(* Logix 5000 project; controller Joltek_RA_5069PLC002 vendor 1 type 14 code 226 rev 34.15; software revision 34.04; part 2 of 3 *)
(* tags used below, declared in another part *)
   CapperData : UDT_MachineData;
   CasePackerData : UDT_MachineData;
   FillerData : UDT_MachineData;
   LabelerData : UDT_MachineData;
   PalletizerData : UDT_MachineData;
   shiftHour : INT;
   HMI_INT : INT[100];
   HMI_REAL : REAL[100];
   Sys_DINT : DINT[100];
   Sys_FIFO_C : CONTROL[50];
   Sys_Timer : TIMER[100];
   System_Date_Time : DINT[7];
(* MainProgram, continued *)

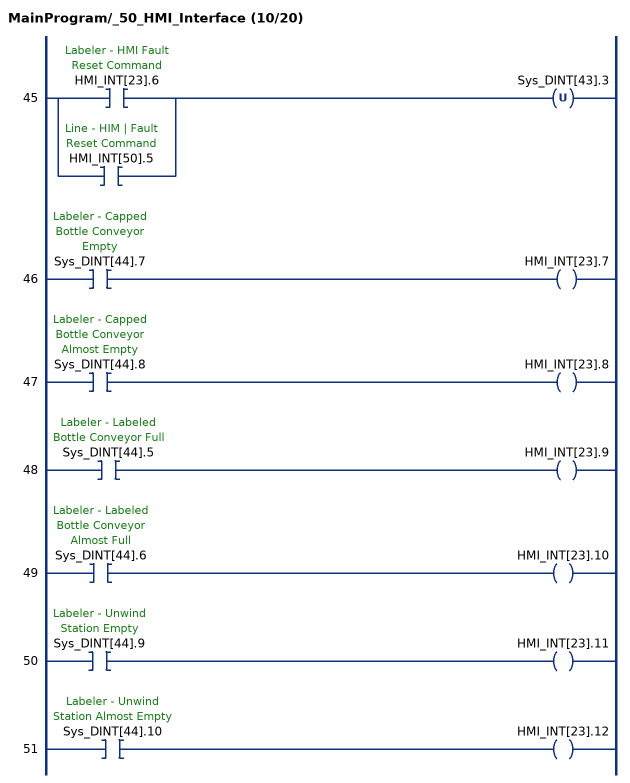
   45: [XIC(HMI_INT[23].6) ,XIC(HMI_INT[50].5) ]OTU(Sys_DINT[43].3);
   46: XIC(Sys_DINT[44].7)OTE(HMI_INT[23].7);
   47: XIC(Sys_DINT[44].8)OTE(HMI_INT[23].8);
   48: XIC(Sys_DINT[44].5)OTE(HMI_INT[23].9);
   49: XIC(Sys_DINT[44].6)OTE(HMI_INT[23].10);
   50: XIC(Sys_DINT[44].9)OTE(HMI_INT[23].11);
   51: XIC(Sys_DINT[44].10)OTE(HMI_INT[23].12);
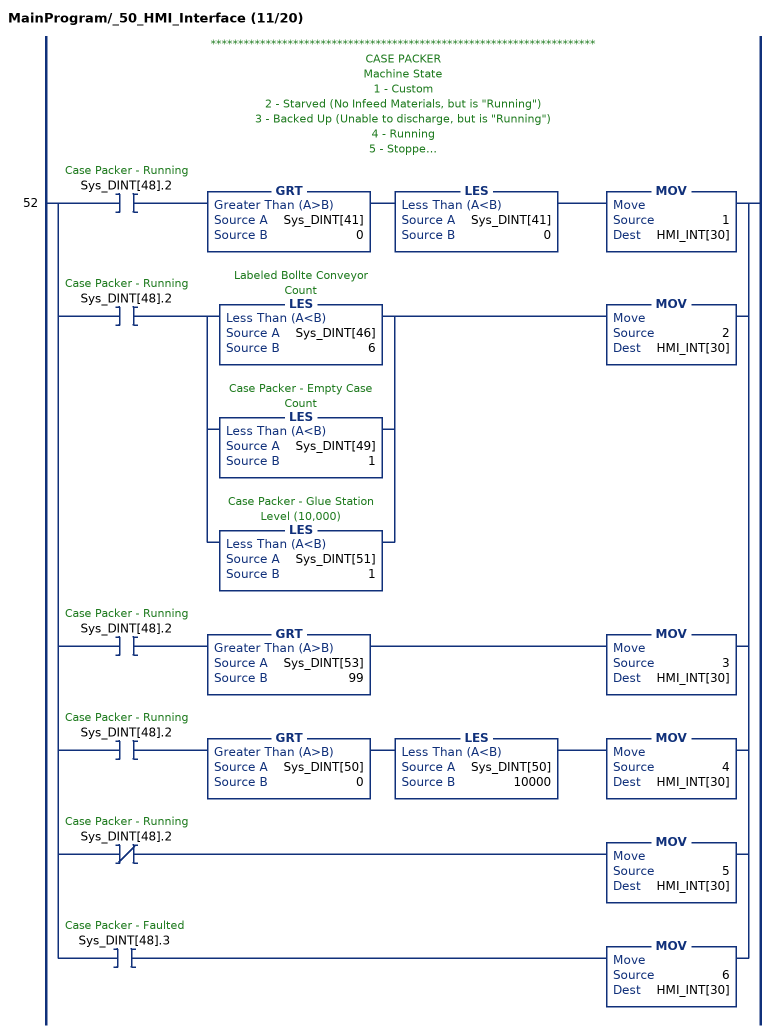
   // **********************************************************************
   // CASE PACKER
   // Machine State
   // 1 - Custom
   // 2 - Starved (No Infeed Materials, but is "Running")
   // 3 - Backed Up (Unable to discharge, but is "Running")
   // 4 - Running
   // 5 - Stopped
   // 6 - Faulted
   52: [XIC(Sys_DINT[48].2) GRT(Sys_DINT[41],0) LES(Sys_DINT[41],0) MOV(1,HMI_INT[30]) ,XIC(Sys_DINT[48].2) [LES(Sys_DINT[46],6) ,LES(Sys_DINT[49],1) ,LES(Sys_DINT[51],1) ] MOV(2,HMI_INT[30]) ,XIC(Sys_DINT[48].2) GRT(Sys_DINT[53],99) MOV(3,HMI_INT[30]) ,XIC(Sys_DINT[48].2) GRT(Sys_DINT[50],0) LES(Sys_DINT[50],10000) MOV(4,HMI_INT[30]) ,XIO(Sys_DINT[48].2) MOV(5,HMI_INT[30]) ,XIC(Sys_DINT[48].3) MOV(6,HMI_INT[30]) ];
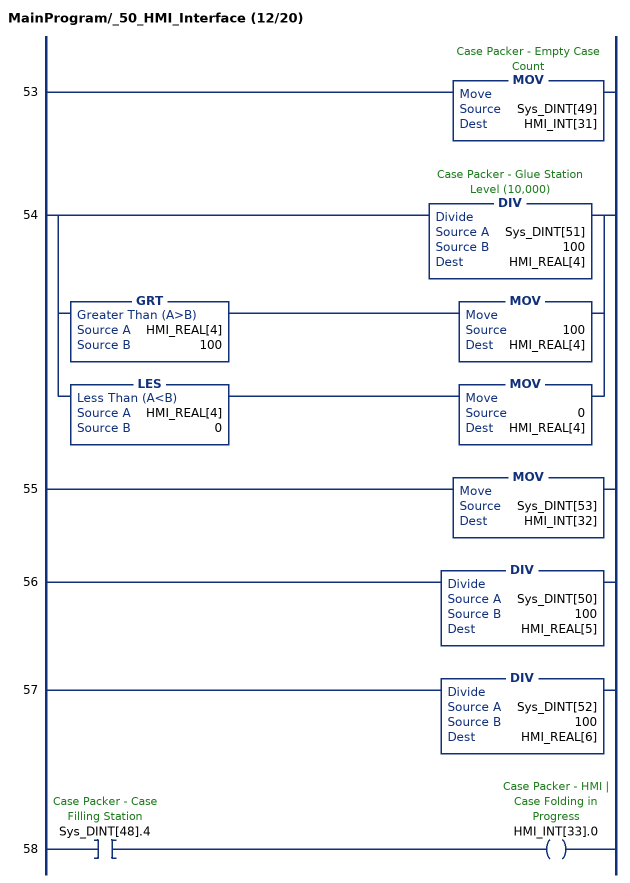
   53: MOV(Sys_DINT[49],HMI_INT[31]);
   54: [DIV(Sys_DINT[51],100,HMI_REAL[4]) ,GRT(HMI_REAL[4],100) MOV(100,HMI_REAL[4]) ,LES(HMI_REAL[4],0) MOV(0,HMI_REAL[4]) ];
   55: MOV(Sys_DINT[53],HMI_INT[32]);
   56: DIV(Sys_DINT[50],100,HMI_REAL[5]);
   57: DIV(Sys_DINT[52],100,HMI_REAL[6]);
   58: XIC(Sys_DINT[48].4)OTE(HMI_INT[33].0);
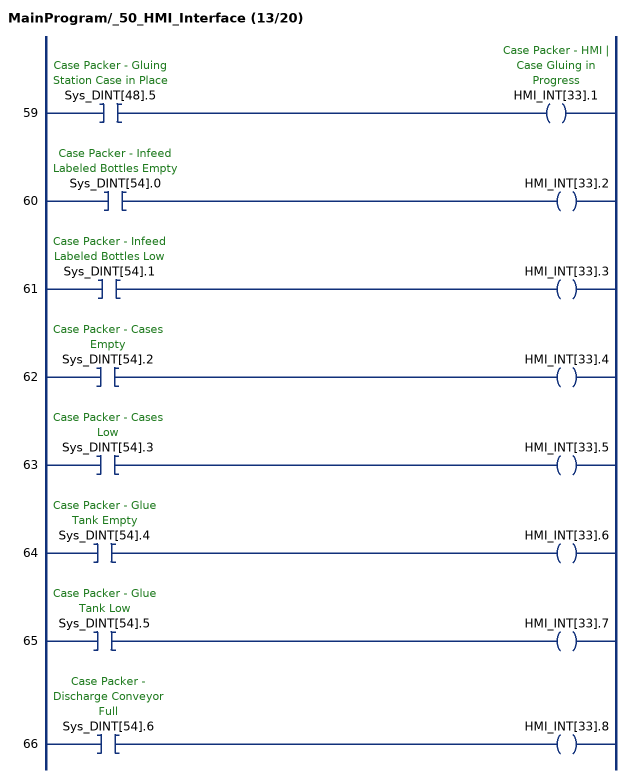
   59: XIC(Sys_DINT[48].5)OTE(HMI_INT[33].1);
   60: XIC(Sys_DINT[54].0)OTE(HMI_INT[33].2);
   61: XIC(Sys_DINT[54].1)OTE(HMI_INT[33].3);
   62: XIC(Sys_DINT[54].2)OTE(HMI_INT[33].4);
   63: XIC(Sys_DINT[54].3)OTE(HMI_INT[33].5);
   64: XIC(Sys_DINT[54].4)OTE(HMI_INT[33].6);
   65: XIC(Sys_DINT[54].5)OTE(HMI_INT[33].7);
   66: XIC(Sys_DINT[54].6)OTE(HMI_INT[33].8);
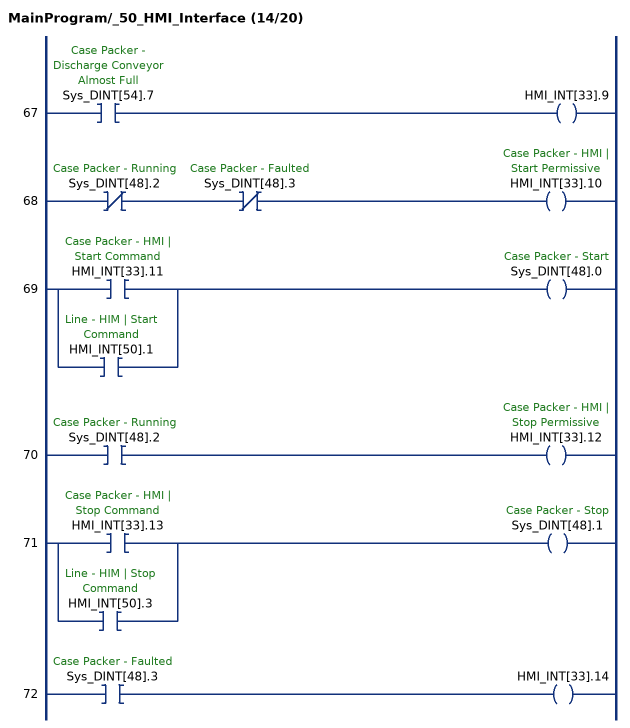
   67: XIC(Sys_DINT[54].7)OTE(HMI_INT[33].9);
   68: XIO(Sys_DINT[48].2)XIO(Sys_DINT[48].3)OTE(HMI_INT[33].10);
   69: [XIC(HMI_INT[33].11) ,XIC(HMI_INT[50].1) ]OTE(Sys_DINT[48].0);
   70: XIC(Sys_DINT[48].2)OTE(HMI_INT[33].12);
   71: [XIC(HMI_INT[33].13) ,XIC(HMI_INT[50].3) ]OTE(Sys_DINT[48].1);
   72: XIC(Sys_DINT[48].3)OTE(HMI_INT[33].14);
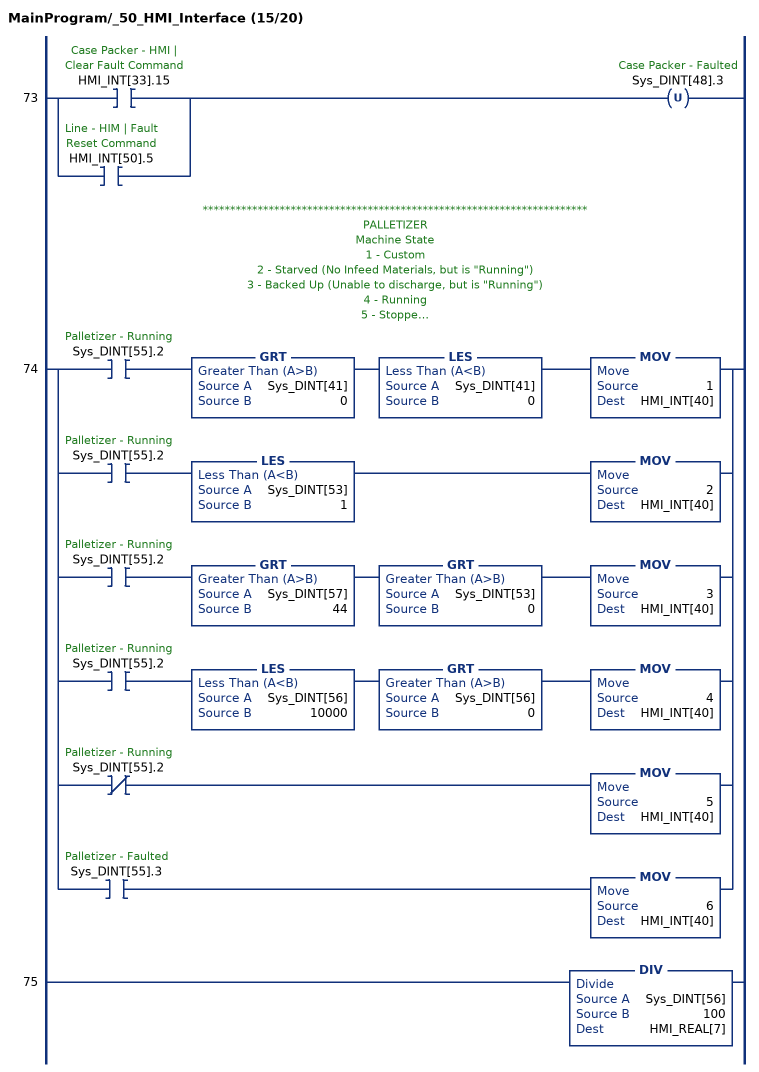
   73: [XIC(HMI_INT[33].15) ,XIC(HMI_INT[50].5) ]OTU(Sys_DINT[48].3);
   // **********************************************************************
   // PALLETIZER
   // Machine State
   // 1 - Custom
   // 2 - Starved (No Infeed Materials, but is "Running")
   // 3 - Backed Up (Unable to discharge, but is "Running")
   // 4 - Running
   // 5 - Stopped
   // 6 - Faulted
   74: [XIC(Sys_DINT[55].2) GRT(Sys_DINT[41],0) LES(Sys_DINT[41],0) MOV(1,HMI_INT[40]) ,XIC(Sys_DINT[55].2) LES(Sys_DINT[53],1) MOV(2,HMI_INT[40]) ,XIC(Sys_DINT[55].2) GRT(Sys_DINT[57],44) GRT(Sys_DINT[53],0) MOV(3,HMI_INT[40]) ,XIC(Sys_DINT[55].2) LES(Sys_DINT[56],10000) GRT(Sys_DINT[56],0) MOV(4,HMI_INT[40]) ,XIO(Sys_DINT[55].2) MOV(5,HMI_INT[40]) ,XIC(Sys_DINT[55].3) MOV(6,HMI_INT[40]) ];
   75: DIV(Sys_DINT[56],100,HMI_REAL[7]);
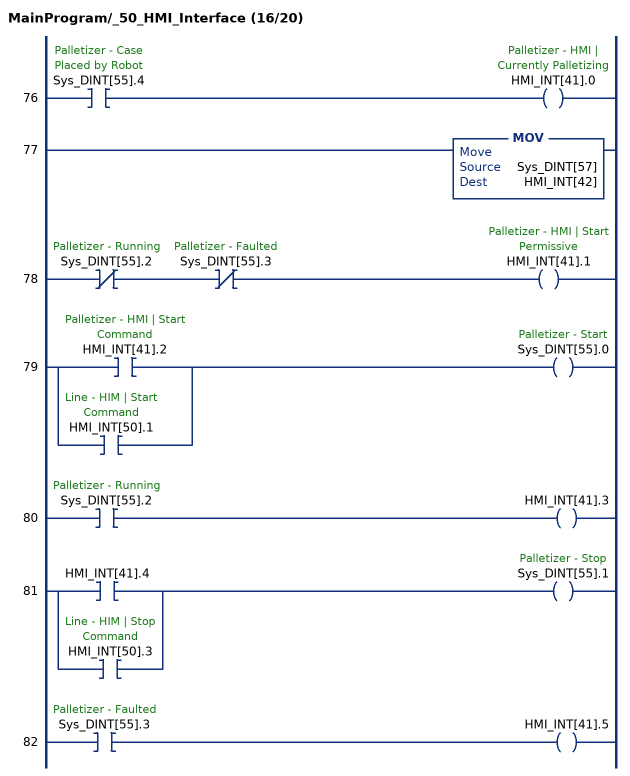
   76: XIC(Sys_DINT[55].4)OTE(HMI_INT[41].0);
   77: MOV(Sys_DINT[57],HMI_INT[42]);
   78: XIO(Sys_DINT[55].2)XIO(Sys_DINT[55].3)OTE(HMI_INT[41].1);
   79: [XIC(HMI_INT[41].2) ,XIC(HMI_INT[50].1) ]OTE(Sys_DINT[55].0);
   80: XIC(Sys_DINT[55].2)OTE(HMI_INT[41].3);
   81: [XIC(HMI_INT[41].4) ,XIC(HMI_INT[50].3) ]OTE(Sys_DINT[55].1);
   82: XIC(Sys_DINT[55].3)OTE(HMI_INT[41].5);
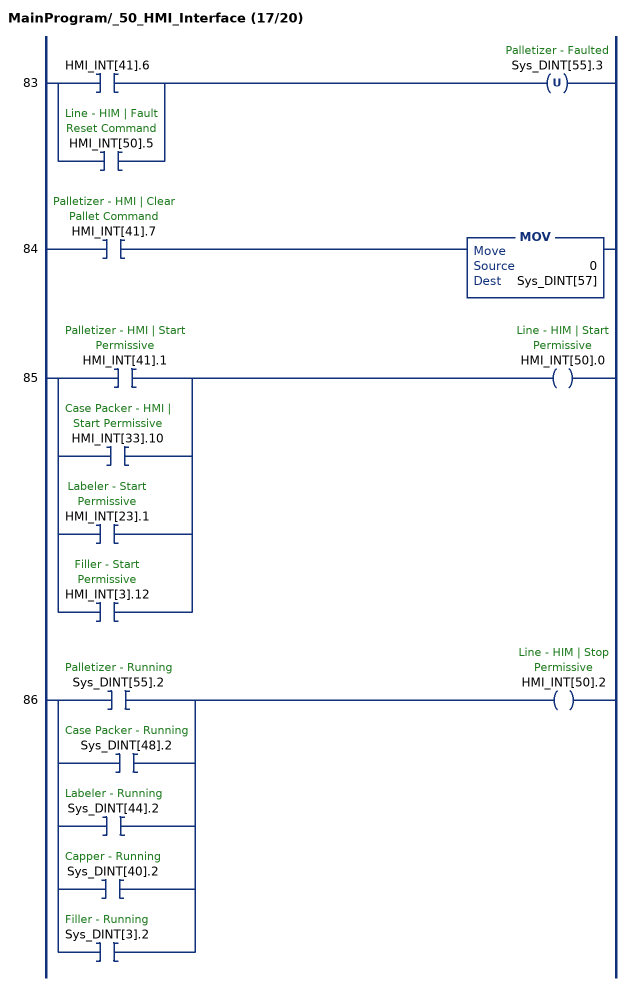
   83: [XIC(HMI_INT[41].6) ,XIC(HMI_INT[50].5) ]OTU(Sys_DINT[55].3);
   84: XIC(HMI_INT[41].7)MOV(0,Sys_DINT[57]);
   85: [XIC(HMI_INT[41].1) ,XIC(HMI_INT[33].10) ,XIC(HMI_INT[23].1) ,XIC(HMI_INT[3].12) ]OTE(HMI_INT[50].0);
   86: [XIC(Sys_DINT[55].2) ,XIC(Sys_DINT[48].2) ,XIC(Sys_DINT[44].2) ,XIC(Sys_DINT[40].2) ,XIC(Sys_DINT[3].2) ]OTE(HMI_INT[50].2);
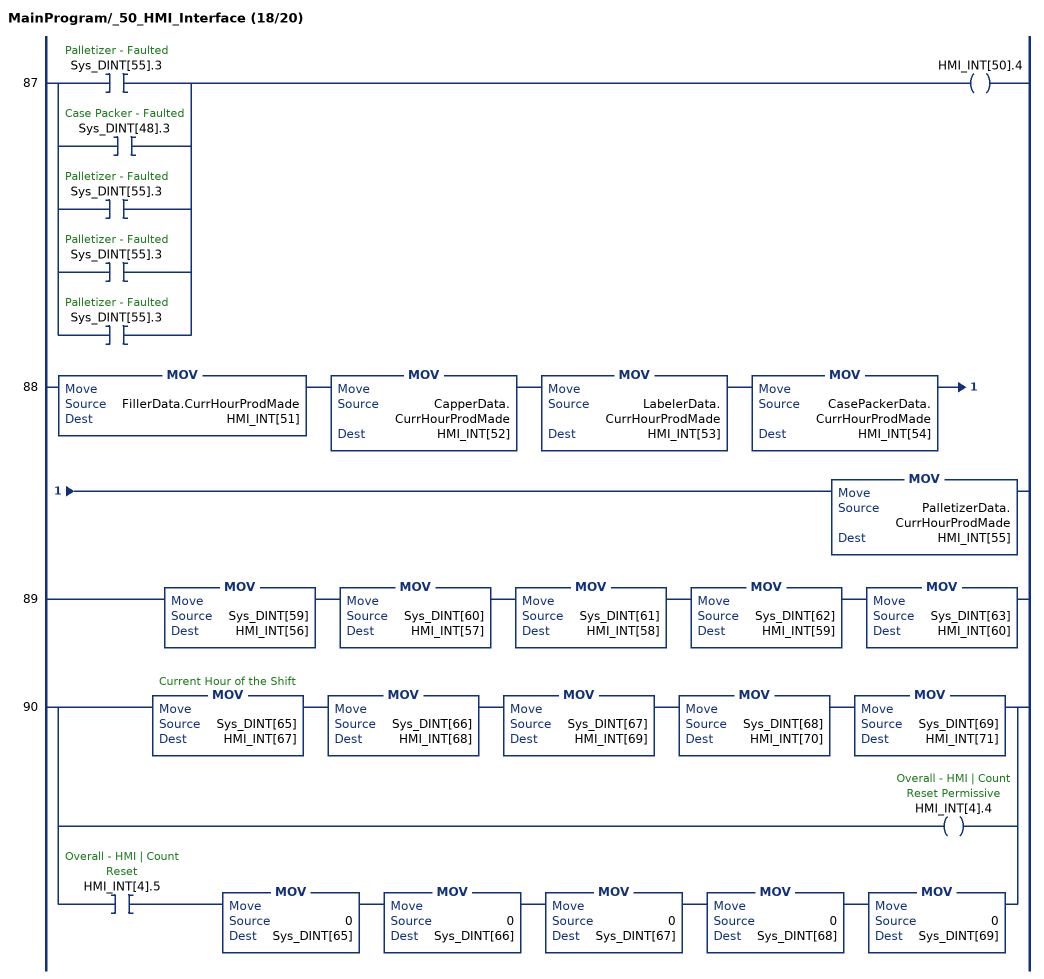
   87: [XIC(Sys_DINT[55].3) ,XIC(Sys_DINT[48].3) ,XIC(Sys_DINT[55].3) ,XIC(Sys_DINT[55].3) ,XIC(Sys_DINT[55].3) ]OTE(HMI_INT[50].4);
   88: MOV(FillerData.CurrHourProdMade,HMI_INT[51])MOV(CapperData.CurrHourProdMade,HMI_INT[52])MOV(LabelerData.CurrHourProdMade,HMI_INT[53])MOV(CasePackerData.CurrHourProdMade,HMI_INT[54])MOV(PalletizerData.CurrHourProdMade,HMI_INT[55]);
   89: MOV(Sys_DINT[59],HMI_INT[56])MOV(Sys_DINT[60],HMI_INT[57])MOV(Sys_DINT[61],HMI_INT[58])MOV(Sys_DINT[62],HMI_INT[59])MOV(Sys_DINT[63],HMI_INT[60]);
   90: [MOV(Sys_DINT[65],HMI_INT[67]) MOV(Sys_DINT[66],HMI_INT[68]) MOV(Sys_DINT[67],HMI_INT[69]) MOV(Sys_DINT[68],HMI_INT[70]) MOV(Sys_DINT[69],HMI_INT[71]) ,OTE(HMI_INT[4].4) ,XIC(HMI_INT[4].5) MOV(0,Sys_DINT[65]) MOV(0,Sys_DINT[66]) MOV(0,Sys_DINT[67]) MOV(0,Sys_DINT[68]) MOV(0,Sys_DINT[69]) ];
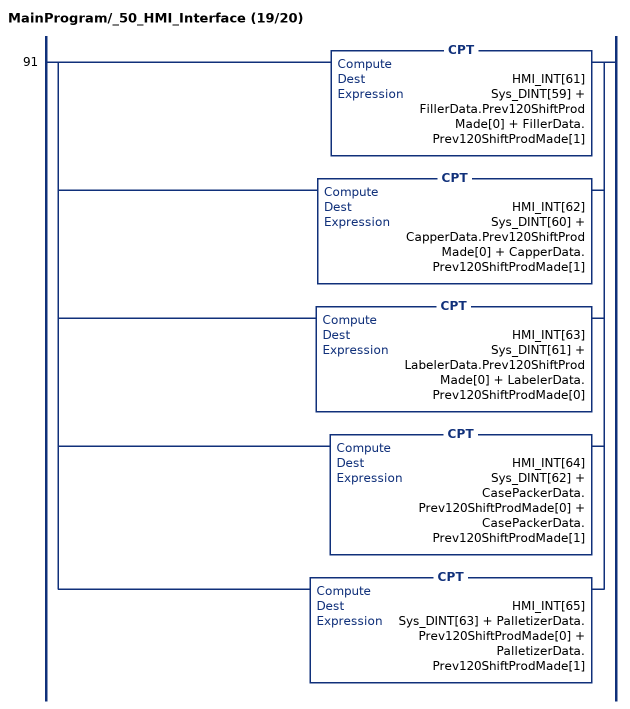
   91: [CPT(HMI_INT[61],Sys_DINT[59] + FillerData.Prev120ShiftProdMade[0] + FillerData.Prev120ShiftProdMade[1]) ,CPT(HMI_INT[62],Sys_DINT[60] + CapperData.Prev120ShiftProdMade[0] + CapperData.Prev120ShiftProdMade[1]) ,CPT(HMI_INT[63],Sys_DINT[61] + LabelerData.Prev120ShiftProdMade[0] + LabelerData.Prev120ShiftProdMade[0]) ,CPT(HMI_INT[64],Sys_DINT[62] + CasePackerData.Prev120ShiftProdMade[0] + CasePackerData.Prev120ShiftProdMade[1]) ,CPT(HMI_INT[65],Sys_DINT[63] + PalletizerData.Prev120ShiftProdMade[0] + PalletizerData.Prev120ShiftProdMade[1]) ];
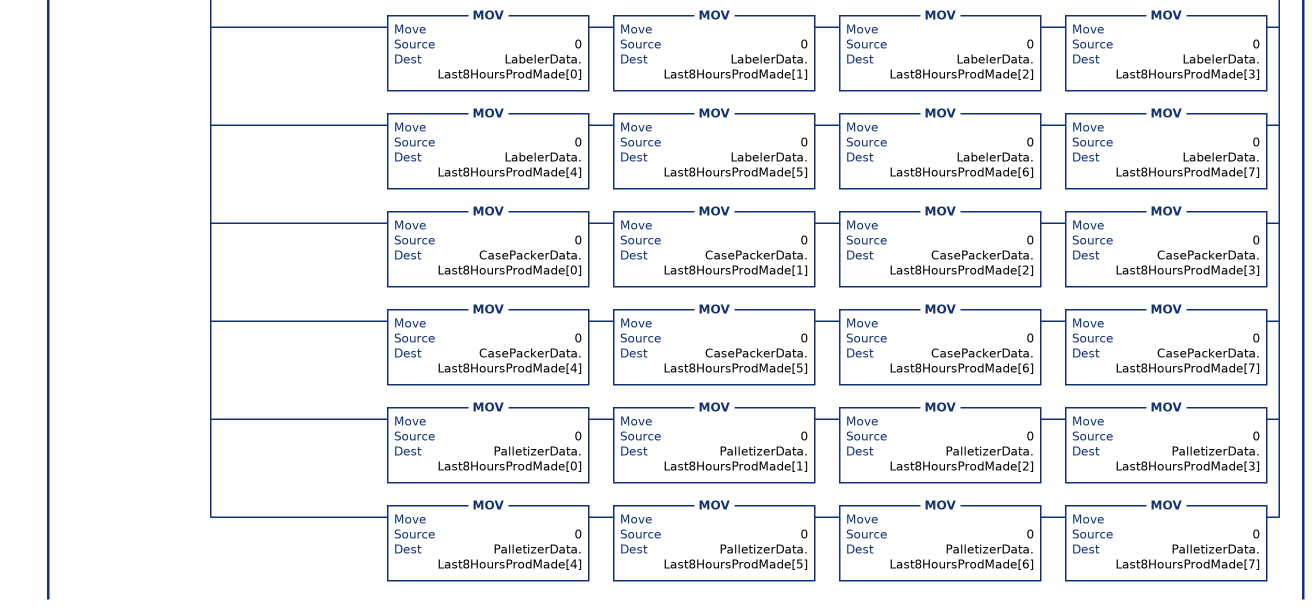
   92: [OTE(HMI_INT[4].6) ,XIC(HMI_INT[4].7) [MOV(0,Sys_DINT[65]) MOV(0,Sys_DINT[66]) MOV(0,Sys_DINT[67]) MOV(0,Sys_DINT[68]) MOV(0,Sys_DINT[69]) ,MOV(0,FillerData.CurrHourProdMade) MOV(0,CapperData.CurrHourProdMade) MOV(0,LabelerData.CurrHourProdMade) MOV(0,CasePackerData.CurrHourProdMade) MOV(0,PalletizerData.CurrHourProdMade) ,MOV(0,FillerData.Prev120ShiftProdMade[0]) MOV(0,FillerData.Prev120ShiftProdMade[1]) MOV(0,CapperData.Prev120ShiftProdMade[0]) MOV(0,CapperData.Prev120ShiftProdMade[1]) ,MOV(0,LabelerData.Prev120ShiftProdMade[0]) MOV(0,LabelerData.Prev120ShiftProdMade[1]) MOV(0,CasePackerData.Prev120ShiftProdMade[0]) MOV(0,CasePackerData.Prev120ShiftProdMade[1]) ,MOV(0,PalletizerData.Prev120ShiftProdMade[0]) MOV(0,PalletizerData.Prev120ShiftProdMade[1]) ,MOV(0,Sys_FIFO_C[1].POS) MOV(0,Sys_FIFO_C[2].POS) MOV(0,Sys_FIFO_C[3].POS) MOV(0,Sys_FIFO_C[4].POS) MOV(0,Sys_FIFO_C[5].POS) ,MOV(0,FillerData.Last8HoursProdMade[0]) MOV(0,FillerData.Last8HoursProdMade[1]) MOV(0,FillerData.Last8HoursProdMade[2]) MOV(0,FillerData.Last8HoursProdMade[3]) ,MOV(0,FillerData.Last8HoursProdMade[4]) MOV(0,FillerData.Last8HoursProdMade[5]) MOV(0,FillerData.Last8HoursProdMade[6]) MOV(0,FillerData.Last8HoursProdMade[7]) ,MOV(0,CapperData.Last8HoursProdMade[0]) MOV(0,CapperData.Last8HoursProdMade[1]) MOV(0,CapperData.Last8HoursProdMade[2]) MOV(0,CapperData.Last8HoursProdMade[3]) ,MOV(0,CapperData.Last8HoursProdMade[4]) MOV(0,CapperData.Last8HoursProdMade[5]) MOV(0,CapperData.Last8HoursProdMade[6]) MOV(0,CapperData.Last8HoursProdMade[7]) ,MOV(0,LabelerData.Last8HoursProdMade[0]) MOV(0,LabelerData.Last8HoursProdMade[1]) MOV(0,LabelerData.Last8HoursProdMade[2]) MOV(0,LabelerData.Last8HoursProdMade[3]) ,MOV(0,LabelerData.Last8HoursProdMade[4]) MOV(0,LabelerData.Last8HoursProdMade[5]) MOV(0,LabelerData.Last8HoursProdMade[6]) MOV(0,LabelerData.Last8HoursProdMade[7]) ,MOV(0,CasePackerData.Last8HoursProdMade[0]) MOV(0,CasePackerData.Last8HoursProdMade[1]) MOV(0,CasePackerData.Last8HoursProdMade[2]) MOV(0,CasePackerData.Last8HoursProdMade[3]) ,MOV(0,CasePackerData.Last8HoursProdMade[4]) MOV(0,CasePackerData.Last8HoursProdMade[5]) MOV(0,CasePackerData.Last8HoursProdMade[6]) MOV(0,CasePackerData.Last8HoursProdMade[7]) ,MOV(0,PalletizerData.Last8HoursProdMade[0]) MOV(0,PalletizerData.Last8HoursProdMade[1]) MOV(0,PalletizerData.Last8HoursProdMade[2]) MOV(0,PalletizerData.Last8HoursProdMade[3]) ,MOV(0,PalletizerData.Last8HoursProdMade[4]) MOV(0,PalletizerData.Last8HoursProdMade[5]) MOV(0,PalletizerData.Last8HoursProdMade[6]) MOV(0,PalletizerData.Last8HoursProdMade[7]) ] ];
END_ROUTINE

ROUTINE _60_DataProcessing   (* ladder *)
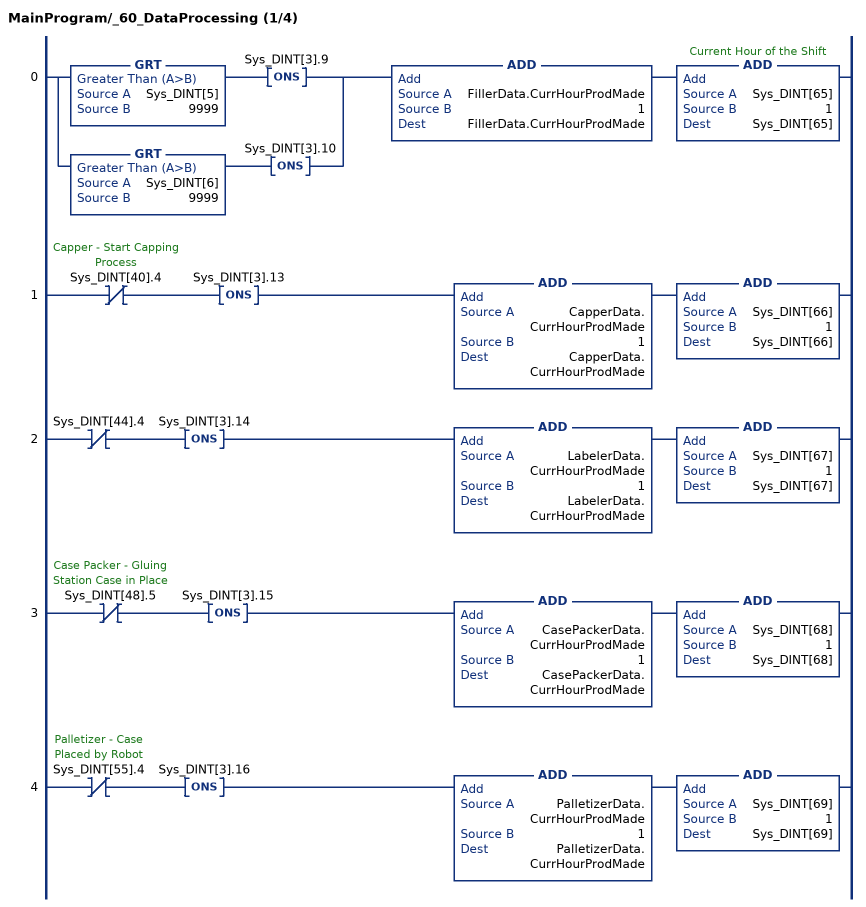
   0: [GRT(Sys_DINT[5],9999) ONS(Sys_DINT[3].9) ,GRT(Sys_DINT[6],9999) ONS(Sys_DINT[3].10) ]ADD(FillerData.CurrHourProdMade,1,FillerData.CurrHourProdMade)ADD(Sys_DINT[65],1,Sys_DINT[65]);
   1: XIO(Sys_DINT[40].4)ONS(Sys_DINT[3].13)ADD(CapperData.CurrHourProdMade,1,CapperData.CurrHourProdMade)ADD(Sys_DINT[66],1,Sys_DINT[66]);
   2: XIO(Sys_DINT[44].4)ONS(Sys_DINT[3].14)ADD(LabelerData.CurrHourProdMade,1,LabelerData.CurrHourProdMade)ADD(Sys_DINT[67],1,Sys_DINT[67]);
   3: XIO(Sys_DINT[48].5)ONS(Sys_DINT[3].15)ADD(CasePackerData.CurrHourProdMade,1,CasePackerData.CurrHourProdMade)ADD(Sys_DINT[68],1,Sys_DINT[68]);
   4: XIO(Sys_DINT[55].4)ONS(Sys_DINT[3].16)ADD(PalletizerData.CurrHourProdMade,1,PalletizerData.CurrHourProdMade)ADD(Sys_DINT[69],1,Sys_DINT[69]);
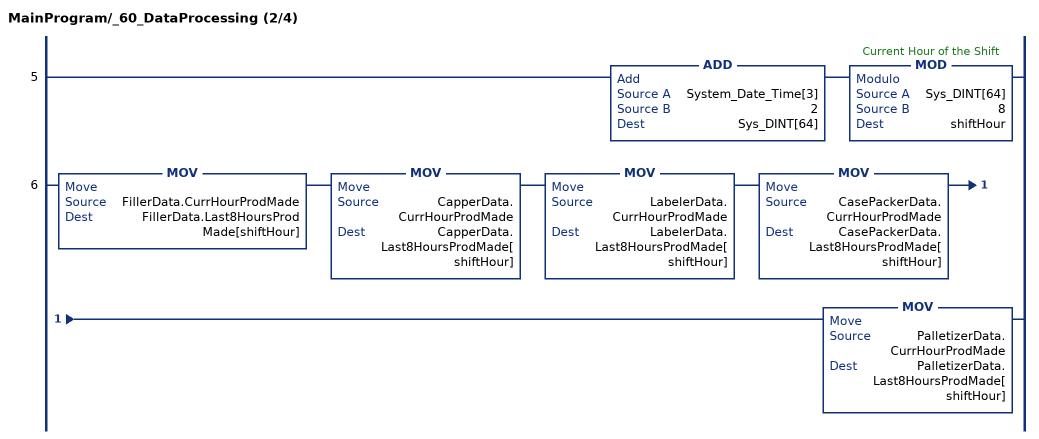
   5: ADD(System_Date_Time[3],2,Sys_DINT[64])MOD(Sys_DINT[64],8,shiftHour);
   6: MOV(FillerData.CurrHourProdMade,FillerData.Last8HoursProdMade[shiftHour])MOV(CapperData.CurrHourProdMade,CapperData.Last8HoursProdMade[shiftHour])MOV(LabelerData.CurrHourProdMade,LabelerData.Last8HoursProdMade[shiftHour])MOV(CasePackerData.CurrHourProdMade,CasePackerData.Last8HoursProdMade[shiftHour])MOV(PalletizerData.CurrHourProdMade,PalletizerData.Last8HoursProdMade[shiftHour]);
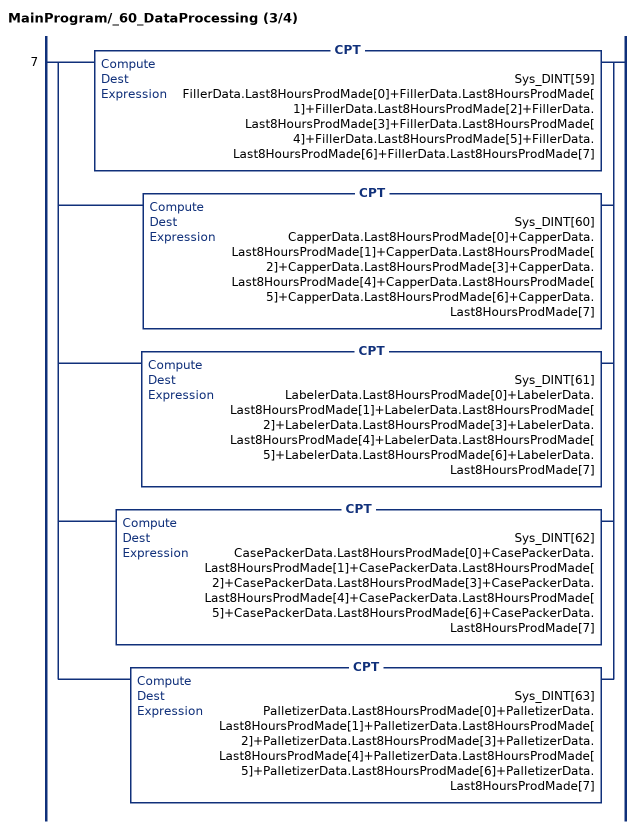
   7: [CPT(Sys_DINT[59],FillerData.Last8HoursProdMade[0]+FillerData.Last8HoursProdMade[1]+FillerData.Last8HoursProdMade[2]+FillerData.Last8HoursProdMade[3]+FillerData.Last8HoursProdMade[4]+FillerData.Last8HoursProdMade[5]+FillerData.Last8HoursProdMade[6]+FillerData.Last8HoursProdMade[7]) ,CPT(Sys_DINT[60],CapperData.Last8HoursProdMade[0]+CapperData.Last8HoursProdMade[1]+CapperData.Last8HoursProdMade[2]+CapperData.Last8HoursProdMade[3]+CapperData.Last8HoursProdMade[4]+CapperData.Last8HoursProdMade[5]+CapperData.Last8HoursProdMade[6]+CapperData.Last8HoursProdMade[7]) ,CPT(Sys_DINT[61],LabelerData.Last8HoursProdMade[0]+LabelerData.Last8HoursProdMade[1]+LabelerData.Last8HoursProdMade[2]+LabelerData.Last8HoursProdMade[3]+LabelerData.Last8HoursProdMade[4]+LabelerData.Last8HoursProdMade[5]+LabelerData.Last8HoursProdMade[6]+LabelerData.Last8HoursProdMade[7]) ,CPT(Sys_DINT[62],CasePackerData.Last8HoursProdMade[0]+CasePackerData.Last8HoursProdMade[1]+CasePackerData.Last8HoursProdMade[2]+CasePackerData.Last8HoursProdMade[3]+CasePackerData.Last8HoursProdMade[4]+CasePackerData.Last8HoursProdMade[5]+CasePackerData.Last8HoursProdMade[6]+CasePackerData.Last8HoursProdMade[7]) ,CPT(Sys_DINT[63],PalletizerData.Last8HoursProdMade[0]+PalletizerData.Last8HoursProdMade[1]+PalletizerData.Last8HoursProdMade[2]+PalletizerData.Last8HoursProdMade[3]+PalletizerData.Last8HoursProdMade[4]+PalletizerData.Last8HoursProdMade[5]+PalletizerData.Last8HoursProdMade[6]+PalletizerData.Last8HoursProdMade[7]) ];
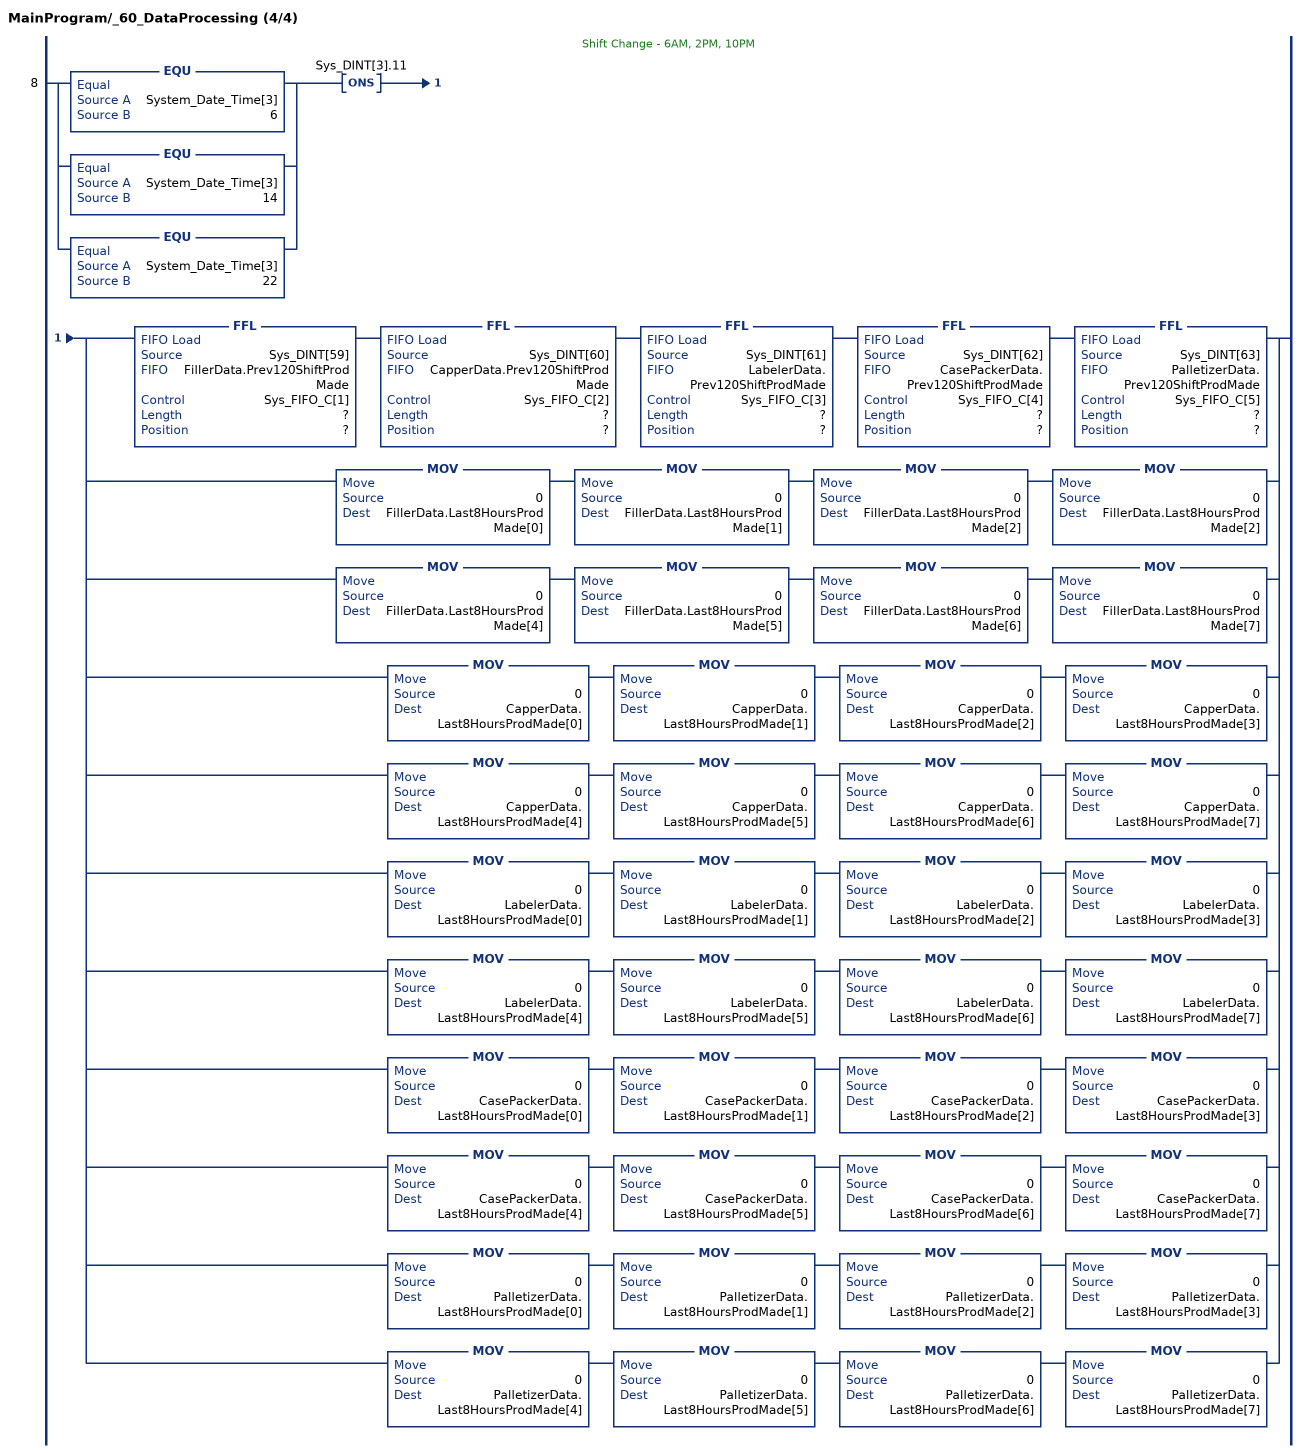
   // Shift Change - 6AM, 2PM, 10PM
   8: [EQU(System_Date_Time[3],6) ,EQU(System_Date_Time[3],14) ,EQU(System_Date_Time[3],22) ]ONS(Sys_DINT[3].11)[FFL(Sys_DINT[59],FillerData.Prev120ShiftProdMade,Sys_FIFO_C[1],?,?) FFL(Sys_DINT[60],CapperData.Prev120ShiftProdMade,Sys_FIFO_C[2],?,?) FFL(Sys_DINT[61],LabelerData.Prev120ShiftProdMade,Sys_FIFO_C[3],?,?) FFL(Sys_DINT[62],CasePackerData.Prev120ShiftProdMade,Sys_FIFO_C[4],?,?) FFL(Sys_DINT[63],PalletizerData.Prev120ShiftProdMade,Sys_FIFO_C[5],?,?) ,MOV(0,FillerData.Last8HoursProdMade[0]) MOV(0,FillerData.Last8HoursProdMade[1]) MOV(0,FillerData.Last8HoursProdMade[2]) MOV(0,FillerData.Last8HoursProdMade[2]) ,MOV(0,FillerData.Last8HoursProdMade[4]) MOV(0,FillerData.Last8HoursProdMade[5]) MOV(0,FillerData.Last8HoursProdMade[6]) MOV(0,FillerData.Last8HoursProdMade[7]) ,MOV(0,CapperData.Last8HoursProdMade[0]) MOV(0,CapperData.Last8HoursProdMade[1]) MOV(0,CapperData.Last8HoursProdMade[2]) MOV(0,CapperData.Last8HoursProdMade[3]) ,MOV(0,CapperData.Last8HoursProdMade[4]) MOV(0,CapperData.Last8HoursProdMade[5]) MOV(0,CapperData.Last8HoursProdMade[6]) MOV(0,CapperData.Last8HoursProdMade[7]) ,MOV(0,LabelerData.Last8HoursProdMade[0]) MOV(0,LabelerData.Last8HoursProdMade[1]) MOV(0,LabelerData.Last8HoursProdMade[2]) MOV(0,LabelerData.Last8HoursProdMade[3]) ,MOV(0,LabelerData.Last8HoursProdMade[4]) MOV(0,LabelerData.Last8HoursProdMade[5]) MOV(0,LabelerData.Last8HoursProdMade[6]) MOV(0,LabelerData.Last8HoursProdMade[7]) ,MOV(0,CasePackerData.Last8HoursProdMade[0]) MOV(0,CasePackerData.Last8HoursProdMade[1]) MOV(0,CasePackerData.Last8HoursProdMade[2]) MOV(0,CasePackerData.Last8HoursProdMade[3]) ,MOV(0,CasePackerData.Last8HoursProdMade[4]) MOV(0,CasePackerData.Last8HoursProdMade[5]) MOV(0,CasePackerData.Last8HoursProdMade[6]) MOV(0,CasePackerData.Last8HoursProdMade[7]) ,MOV(0,PalletizerData.Last8HoursProdMade[0]) MOV(0,PalletizerData.Last8HoursProdMade[1]) MOV(0,PalletizerData.Last8HoursProdMade[2]) MOV(0,PalletizerData.Last8HoursProdMade[3]) ,MOV(0,PalletizerData.Last8HoursProdMade[4]) MOV(0,PalletizerData.Last8HoursProdMade[5]) MOV(0,PalletizerData.Last8HoursProdMade[6]) MOV(0,PalletizerData.Last8HoursProdMade[7]) ];
END_ROUTINE

ROUTINE _98_RandomizerLogic   (* ladder *)
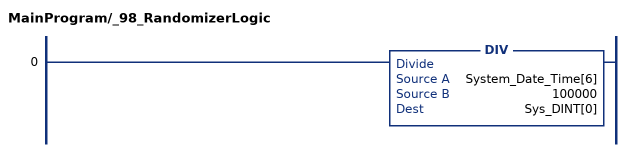
   0: DIV(System_Date_Time[6],100000,Sys_DINT[0]);
END_ROUTINE

ROUTINE _99_TestLogic   (* ladder *)
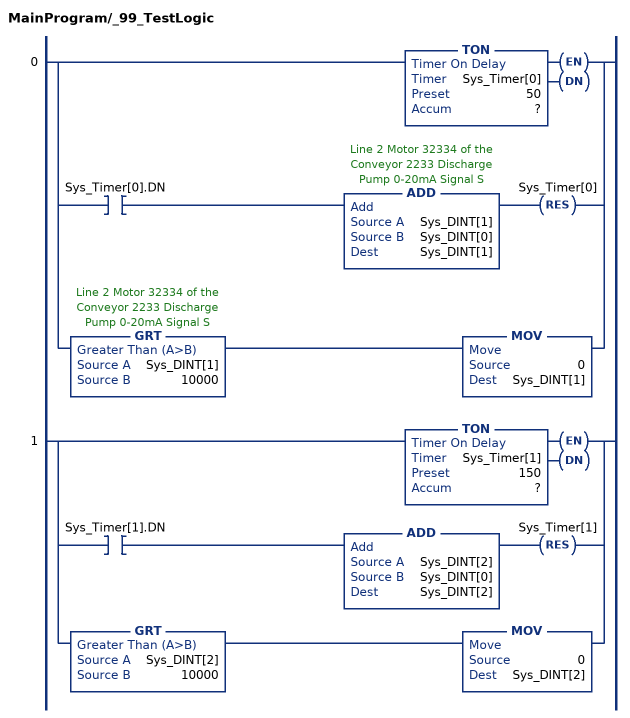
   0: [TON(Sys_Timer[0],?,?) ,XIC(Sys_Timer[0].DN) ADD(Sys_DINT[1],Sys_DINT[0],Sys_DINT[1]) RES(Sys_Timer[0]) ,GRT(Sys_DINT[1],10000) MOV(0,Sys_DINT[1]) ];
   1: [TON(Sys_Timer[1],?,?) ,XIC(Sys_Timer[1].DN) ADD(Sys_DINT[2],Sys_DINT[0],Sys_DINT[2]) RES(Sys_Timer[1]) ,GRT(Sys_DINT[2],10000) MOV(0,Sys_DINT[2]) ];
END_ROUTINE

ROUTINE MainRoutine   (* ladder *)
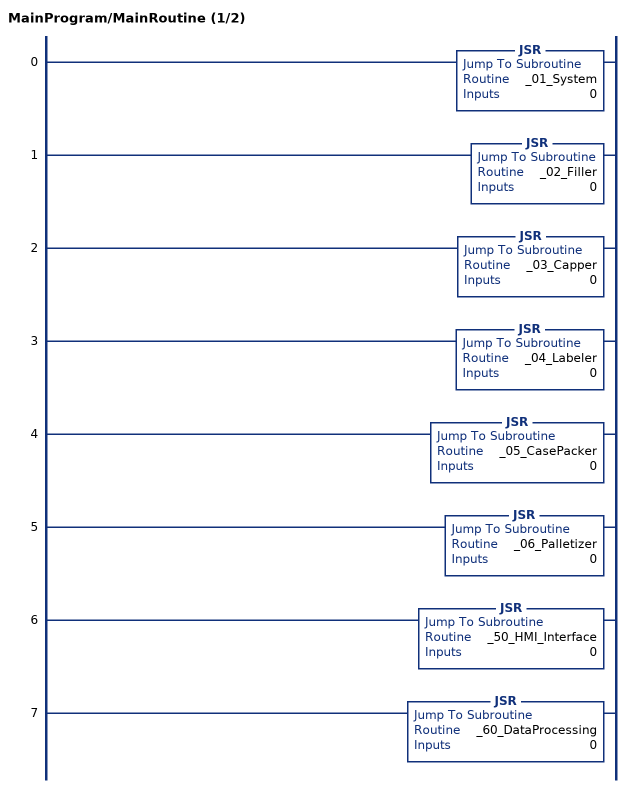
   0: JSR(_01_System,0);
   1: JSR(_02_Filler,0);
   2: JSR(_03_Capper,0);
   3: JSR(_04_Labeler,0);
   4: JSR(_05_CasePacker,0);
   5: JSR(_06_Palletizer,0);
   6: JSR(_50_HMI_Interface,0);
   7: JSR(_60_DataProcessing,0);
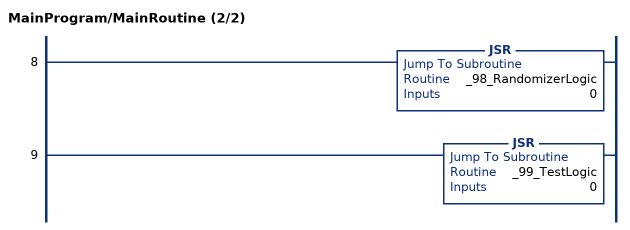
   8: JSR(_98_RandomizerLogic,0);
   9: JSR(_99_TestLogic,0);
END_ROUTINE
END_PROGRAM
